FUNCTION_BLOCK Q_FontAttributes (* Command change font attributes ( Part 6 - F.28 ) *)
  (* Standard: ISO 11783-6; Description: This command is used to change the font attributes in a font attributes object. Return values iso_s16 - E_NO_ERR - OK - E_OVERFLOW - buffer overflow - E_NOACT - Command not possible in current state - E_NO_INSTANCE - No VT client available *)
  (* Version 1.0, 2022-07-08, franz *)
  (* Documentation:
  This command is used to change the font attributes in a font attributes object.
   Return values
   iso_s16
    - E_NO_ERR - OK
   - E_OVERFLOW - buffer overflow
   - E_NOACT - Command not possible in current state
   - E_NO_INSTANCE - No VT client available
  *)
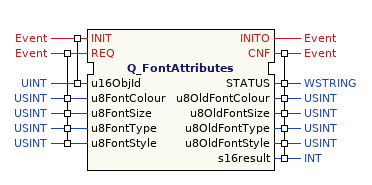
  EVENT_INPUT
    INIT WITH u16ObjId; (* Service Initialization *)
    REQ WITH u8FontColour, u8FontSize, u8FontType, u8FontStyle; (* Service Request *)
  END_EVENT
  EVENT_OUTPUT
    INITO; (* Initialization Confirm *)
    CNF WITH STATUS, u8OldFontType, u8OldFontColour, u8OldFontSize, s16result, u8OldFontStyle; (* Confirmation of Requested Service *)
  END_EVENT
  VAR_INPUT
    u16ObjId : UINT; (* Object ID *)
    u8FontColour : USINT; (* New font colour (see Part 6 - A.3) *)
    u8FontSize : USINT; (* New font size (see Part 6 - B.14) *)
    u8FontType : USINT; (* New font type (see Part 6 - B.14) *)
    u8FontStyle : USINT; (* New font style (see Part 6 - B.14) *)
  END_VAR
  VAR_OUTPUT
    STATUS : WSTRING; (* Service Status *)
    u8OldFontColour : USINT; (* Old font colour (see Part 6 - A.3) *)
    u8OldFontSize : USINT; (* Old font size (see Part 6 - B.14) *)
    u8OldFontType : USINT; (* Old font type (see Part 6 - B.14) *)
    u8OldFontStyle : USINT; (* Old font style (see Part 6 - B.14) *)
    s16result : INT; (* retval see description *)
  END_VAR
END_FUNCTION_BLOCK
